(* CoDeSys 2.3 library: Flexlink V1_0.lib *)
(* Libraries: STANDARD.LIB 5.6.98 12:03:02 *)

(* Global variable list: Global_Variables *)
VAR_GLOBAL
(**************************************************************************************************************)
(* System Bit *)
(**************************************************************************************************************)

	OFF_50ms		: BOOL;
	ON_50ms		: BOOL;
	Clock50msOnPls	: BOOL;
	OFF_100ms		: BOOL;
	ON_100ms		: BOOL;
	Clock100msOnPls	: BOOL;
	OFF_500ms		: BOOL;
	ON_500ms		: BOOL;
	Clock500msOnPls	: BOOL;
	OFF_1s			: BOOL;
	ON_1s			: BOOL;
	Clock1sOnPls	: BOOL;
	Always_ON		:BOOL;
	Always_Off		:BOOL;
	Debug			:BOOL := TRUE;

(**************************************************************************************************************)
(* Machine Standard Word *)
(**************************************************************************************************************)

	ErrorDWord 			AT %MD1000:  ARRAY [0..20,1..10] OF DWORD;
	WarningDWord		AT%MD2000: ARRAY [0..20,1..10] OF DWORD;
	AutoDWord 			AT %MD3000:  ARRAY [0..20,1..10] OF DWORD;
	OriginDWord 			AT %MD4000:  ARRAY [0..20,1..10] OF DWORD;

	InputByte				AT %IB0: ARRAY [0..500] OF BYTE;
	OutputByte			AT %QB0: ARRAY [0..500] OF BYTE;

(**************************************************************************************************************)
(* Machine and Station Control *)
(**************************************************************************************************************)
	MC:Struc_Machine_Ctrl;
	SC :ARRAY[0..20] OF Struc_Station_Ctrl;

(**************************************************************************************************************)
(* Manual Control *)
(**************************************************************************************************************)
	ManualSafetyOK		:BOOL;
	M_StepFwdPls		:BOOL;
	M_StepBwdPls		:BOOL;
	M_StepRun			:BOOL;

(**************************************************************************************************************)
(* Input/Output *)
(**************************************************************************************************************)
	InputWord			AT%IB0	:ARRAY [0..100] OF BOOL;


END_VAR

(* Global variable list: Global_Variables_Error *)
VAR_GLOBAL
	E_EmgStop			: BOOL;
	E_LightCurtain		: BOOL;
	E_AirLow 			: BOOL;
	E_SafetyDoorOpen	: BOOL;
END_VAR

(* Global variable list: Global_Variables_HMI *)
VAR_GLOBAL
	T_AutoRunString:		STRING;

	T_StepRun:			BOOL;
	T_StepStop:			BOOL;
	T_StepBwd:			BOOL;
	T_StepFwd:			BOOL;
	T_StationError:		BOOL;
	T_Origin:				BOOL;
	T_OneCycleRun:		BOOL;
	T_ManualCycleTime:	TIME;
	T_Curr_Step_Station: 	UINT;
	T_EndProd:			BOOL;

	V_StepRunCurrStation:	STRING;
	V_StepRunStatus:		STRING;
	V_AutorunString:		STRING;
END_VAR

(* Global variable list: Global_Variables_Holding *)
VAR_GLOBAL RETAIN
	Password_Control: Std_Password_Ctrl;

(* Parameter Setting *)
	Number_of_Station : INT;

END_VAR

(* Data type *)
TYPE Struc_Hist_Step_Case :
STRUCT
	CurrentStepHist	: INT;
	NextStepHist		: INT;
	StepTime		: TIME;
END_STRUCT
END_TYPE

(* Data type *)
TYPE Struc_Machine_Ctrl :
STRUCT
(* Mode Bit*)
	AutoMode		:BOOL;
	ManualMode		:BOOL;

(* Status Bit*)
	DryRun			:BOOL;
	Stop			:BOOL;
	AutoRunning		:BOOL;
	StopPressed		:BOOL;


	StationStopErr 	:BOOL;
	Warning			:BOOL;
	WarningBuzzer	:BOOL;
	Trouble			:BOOL;
	ErrDetection		:BOOL;


	OriginSchRun		:BOOL;
	InxOrigin			:BOOL;
	AllOrigin			:BOOL;
	AllStationRdy		:BOOL;
	AllStationNoWP 	:BOOL;

END_STRUCT
END_TYPE

(* Data type *)
TYPE Struc_Station_Ctrl :
STRUCT

	Running			:BOOL;
	AutoRun			:BOOL;
	RunReq			:BOOL;		(*Station Start Work Request*)
	Done			:BOOL;		(*Station Work Complete*)
	RunCond		:BOOL;
	Run_NextStepPls	:BOOL;
	Run_PrevStepPls	:BOOL;
	M_Step			:BOOL;

	Origin			:BOOL;   		(* Station Already Origin *)
	Rdy				:BOOL;			(* Station Ready *)
	NoWP 			:BOOL;
	MajorFault		:BOOL;	(* Station Major Fault *)
	MinorFault		:BOOL;	(* Station Minor Fault *)
	Warning			:BOOL;		(* Station Warning *)
	Bypass			:BOOL;		(* Station Bypass *)

	Name			:STRING;
	Status			:STRING;
	CycleTime	:TIME;

END_STRUCT
END_TYPE

(* POU Password_Output, ST *)
PROGRAM Password_Output
VAR

	pls_PasswordOK: R_TRIG;
	PasswordOKPls:BOOL;
END_VAR
(**************************************************************************************************************)
(* HMI Password Control*)
(**************************************************************************************************************)

Password_Control(
	In_PasswordConfig:= '9999');

pls_PasswordOK(CLK:= Password_Control.Out_PasswordOK OR Password_Control.Out_PasswordChanged);
PasswordOKPls := pls_PasswordOK.Q;

IF PasswordOKPls THEN
	CurrentVisu := 'TP40_SETTING';
END_IF
END_PROGRAM

(* POU Std_System_Out, LD *)
PROGRAM Std_System_Out
VAR

	Clk50ms:TON;
	ClkOff50ms:TON;
	Clk100ms:TON;
	ClkOff100ms:TON;
	Clk500ms:TON;
	ClkOff500ms:TON;
	ClkOn1s:TON;
	ClkOff1s:TON;

	T50ms_RTRIG: R_TRIG;
	T100ms_RTRIG: R_TRIG;
	T500ms_RTRIG: R_TRIG;
	T1s_RTRIG: R_TRIG;

END_VAR
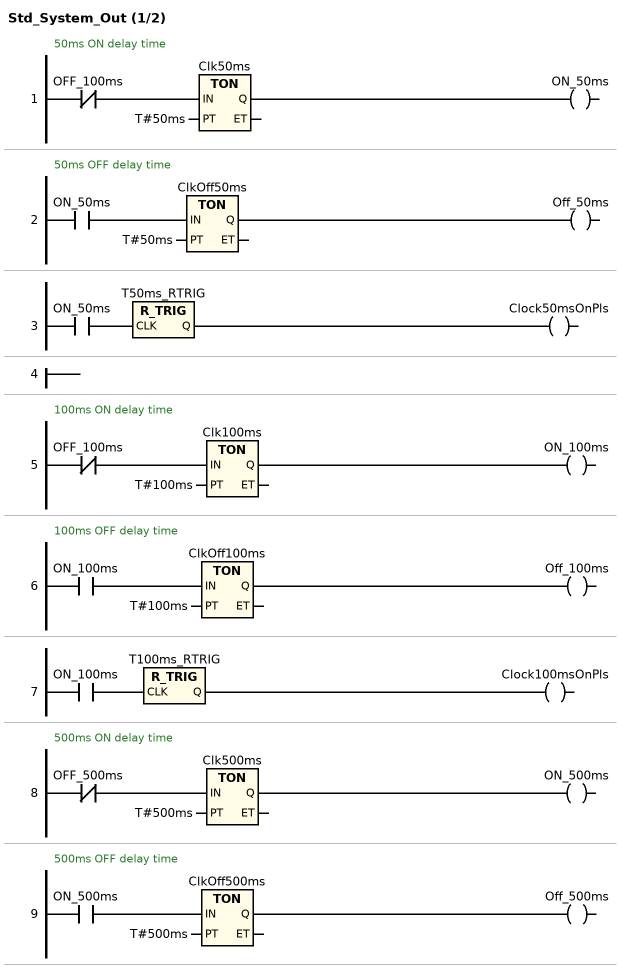
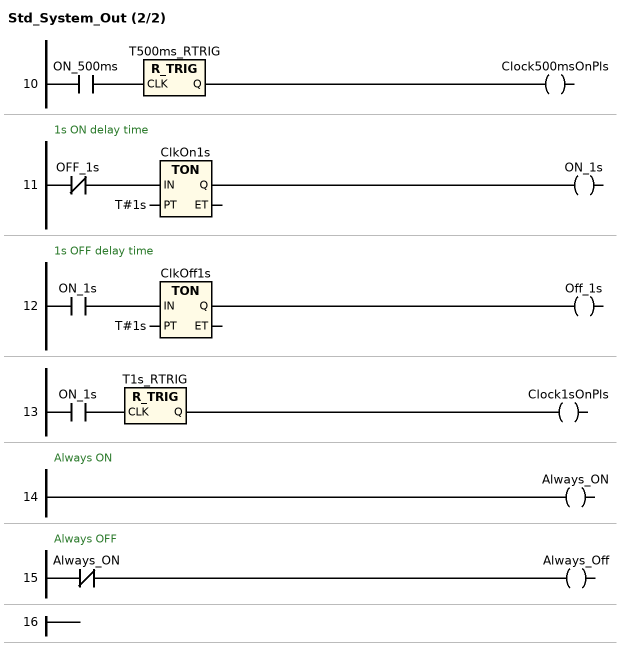
_LD_ (* Ladder Diagram *)
NETWORK 1 (* 50ms ON delay time *)
	[/OFF_100ms] - Clk50ms:TON(IN: *, PT: T#50ms) --- (ON_50ms)
NETWORK 2 (* 50ms OFF delay time *)
	[ON_50ms] - ClkOff50ms:TON(IN: *, PT: T#50ms) --- (Off_50ms)
NETWORK 3
	[ON_50ms] - T50ms_RTRIG:R_TRIG(CLK: *) --- (Clock50msOnPls)
NETWORK 4
	*
NETWORK 5 (* 100ms ON delay time *)
	[/OFF_100ms] - Clk100ms:TON(IN: *, PT: T#100ms) --- (ON_100ms)
NETWORK 6 (* 100ms OFF delay time *)
	[ON_100ms] - ClkOff100ms:TON(IN: *, PT: T#100ms) --- (Off_100ms)
NETWORK 7
	[ON_100ms] - T100ms_RTRIG:R_TRIG(CLK: *) --- (Clock100msOnPls)
NETWORK 8 (* 500ms ON delay time *)
	[/OFF_500ms] - Clk500ms:TON(IN: *, PT: T#500ms) --- (ON_500ms)
NETWORK 9 (* 500ms OFF delay time *)
	[ON_500ms] - ClkOff500ms:TON(IN: *, PT: T#500ms) --- (Off_500ms)
NETWORK 10
	[ON_500ms] - T500ms_RTRIG:R_TRIG(CLK: *) --- (Clock500msOnPls)
NETWORK 11 (* 1s ON delay time *)
	[/OFF_1s] - ClkOn1s:TON(IN: *, PT: T#1s) --- (ON_1s)
NETWORK 12 (* 1s OFF delay time *)
	[ON_1s] - ClkOff1s:TON(IN: *, PT: T#1s) --- (Off_1s)
NETWORK 13
	[ON_1s] - T1s_RTRIG:R_TRIG(CLK: *) --- (Clock1sOnPls)
NETWORK 14 (* Always ON *)
	* --- (Always_ON)
NETWORK 15 (* Always OFF *)
	[/Always_ON] --- (Always_Off)
NETWORK 16
	*
_END_LD_
(* the same logic as Structured Text *)
(* Network 1: 50ms ON delay time *)
Clk50ms(IN := NOT OFF_100ms, PT := T#50ms);
ON_50ms := Clk50ms.Q;
(* Network 2: 50ms OFF delay time *)
ClkOff50ms(IN := ON_50ms, PT := T#50ms);
Off_50ms := ClkOff50ms.Q;
(* Network 3 *)
T50ms_RTRIG(CLK := ON_50ms);
Clock50msOnPls := T50ms_RTRIG.Q;
(* Network 4 *)
(* Network 5: 100ms ON delay time *)
Clk100ms(IN := NOT OFF_100ms, PT := T#100ms);
ON_100ms := Clk100ms.Q;
(* Network 6: 100ms OFF delay time *)
ClkOff100ms(IN := ON_100ms, PT := T#100ms);
Off_100ms := ClkOff100ms.Q;
(* Network 7 *)
T100ms_RTRIG(CLK := ON_100ms);
Clock100msOnPls := T100ms_RTRIG.Q;
(* Network 8: 500ms ON delay time *)
Clk500ms(IN := NOT OFF_500ms, PT := T#500ms);
ON_500ms := Clk500ms.Q;
(* Network 9: 500ms OFF delay time *)
ClkOff500ms(IN := ON_500ms, PT := T#500ms);
Off_500ms := ClkOff500ms.Q;
(* Network 10 *)
T500ms_RTRIG(CLK := ON_500ms);
Clock500msOnPls := T500ms_RTRIG.Q;
(* Network 11: 1s ON delay time *)
ClkOn1s(IN := NOT OFF_1s, PT := T#1s);
ON_1s := ClkOn1s.Q;
(* Network 12: 1s OFF delay time *)
ClkOff1s(IN := ON_1s, PT := T#1s);
Off_1s := ClkOff1s.Q;
(* Network 13 *)
T1s_RTRIG(CLK := ON_1s);
Clock1sOnPls := T1s_RTRIG.Q;
(* Network 14: Always ON *)
Always_ON := TRUE;
(* Network 15: Always OFF *)
Always_Off := NOT Always_ON;
(* Network 16 *)
END_PROGRAM

(* POU Std_Cylinder_Ctrl, LD *)
FUNCTION_BLOCK Std_Cylinder_Ctrl

VAR_INPUT
	IN:BOOL;
	IN_CylName:STRING;
	In_Enable:BOOL;
	In_Reset:BOOL;


	(*Trigger*)
	In_AutoWork:BOOL;
	In_AutoHome:BOOL;
	In_OrgWork:BOOL;
	In_OrgHome:BOOL;
	(*Mechanical Interlock*)
	In_WorkXLock:BOOL;
	In_HomeXLock:BOOL;
	(*Sensors*)
	In_WorkRS:BOOL;
	In_HomeRS:BOOL;

	(*Timer*)
	In_WorkTON:TIME;
	In_HomeTON:TIME;
	in_Timeout:TIME;
END_VAR

VAR_OUTPUT
	Q:BOOL;
	Out_WorkSV:BOOL;
	Out_HomeSV:BOOL;
	E_WorkErr:BOOL;
	E_HomeErr:BOOL;
	S_WorkPos:BOOL;
	S_HomePos:BOOL;
END_VAR

VAR
	(* Trigger*)
	T_ManWork:BOOL;
	T_ManHome:BOOL;

	Loc_Work:BOOL;
	Loc_Home:BOOL;
	Err_Cyl:BOOL;
	Fwd_TOut: TON;
	Bwd_TOut: TON;
	Fwd_TON: TON;
	Bwd_TON: TON;
	Loc_WorkPls: BOOL;
	FwdPls: R_TRIG;
	BwdPls: R_TRIG;
	Loc_HomePls: BOOL;
	Out_RSErr:BOOL;
	FwdPosPls: F_TRIG;
	BwdPosPls: F_TRIG;
END_VAR
VAR_IN_OUT

END_VAR
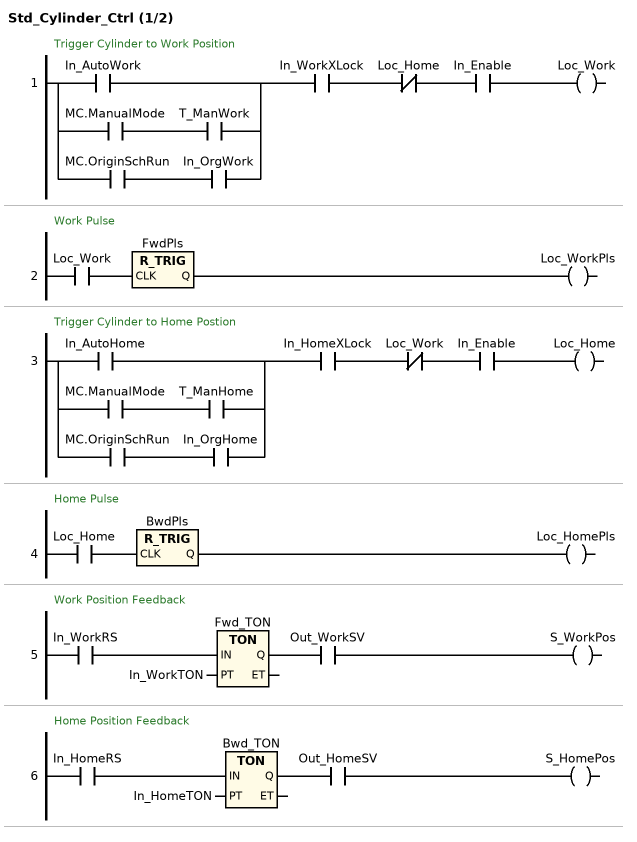
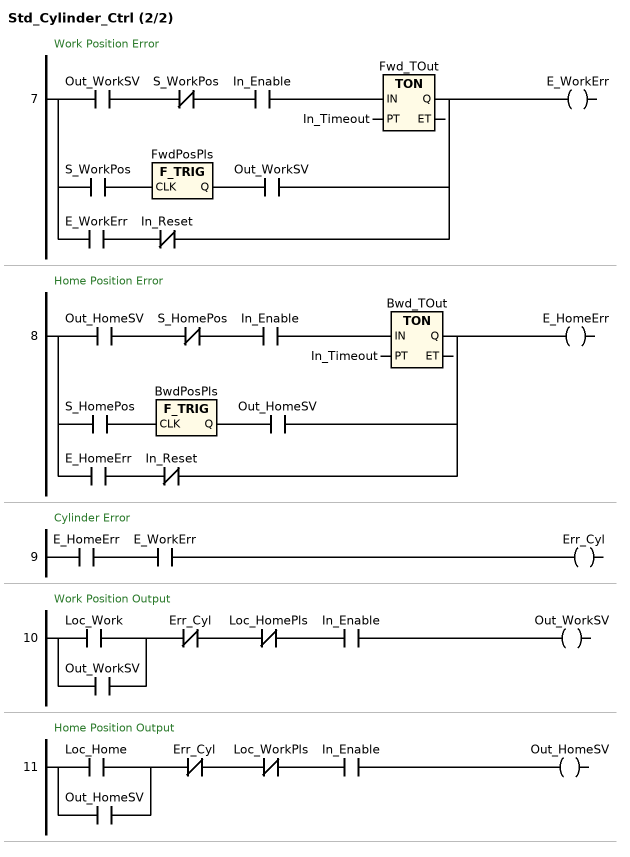
_LD_ (* Ladder Diagram *)
NETWORK 1 (* Trigger Cylinder to Work Position *)
	{ [In_AutoWork] | [MC.ManualMode] - [T_ManWork] | [MC.OriginSchRun] - [In_OrgWork] } - [In_WorkXLock] - [/Loc_Home] - [In_Enable] --- (Loc_Work)
NETWORK 2 (* Work Pulse *)
	[Loc_Work] - FwdPls:R_TRIG(CLK: *) --- (Loc_WorkPls)
NETWORK 3 (* Trigger Cylinder to Home Postion *)
	{ [In_AutoHome] | [MC.ManualMode] - [T_ManHome] | [MC.OriginSchRun] - [In_OrgHome] } - [In_HomeXLock] - [/Loc_Work] - [In_Enable] --- (Loc_Home)
NETWORK 4 (* Home Pulse *)
	[Loc_Home] - BwdPls:R_TRIG(CLK: *) --- (Loc_HomePls)
NETWORK 5 (* Work Position Feedback *)
	[In_WorkRS] - Fwd_TON:TON(IN: *, PT: In_WorkTON) - [Out_WorkSV] --- (S_WorkPos)
NETWORK 6 (* Home Position Feedback *)
	[In_HomeRS] - Bwd_TON:TON(IN: *, PT: In_HomeTON) - [Out_HomeSV] --- (S_HomePos)
NETWORK 7 (* Work Position Error *)
	{ [Out_WorkSV] - [/S_WorkPos] - [In_Enable] - Fwd_TOut:TON(IN: *, PT: In_Timeout) | [S_WorkPos] - FwdPosPls:F_TRIG(CLK: *) - [Out_WorkSV] | [E_WorkErr] - [/In_Reset] } --- (E_WorkErr)
NETWORK 8 (* Home Position Error *)
	{ [Out_HomeSV] - [/S_HomePos] - [In_Enable] - Bwd_TOut:TON(IN: *, PT: In_Timeout) | [S_HomePos] - BwdPosPls:F_TRIG(CLK: *) - [Out_HomeSV] | [E_HomeErr] - [/In_Reset] } --- (E_HomeErr)
NETWORK 9 (* Cylinder Error *)
	[E_HomeErr] - [E_WorkErr] --- (Err_Cyl)
NETWORK 10 (* Work Position Output *)
	{ [Loc_Work] | [Out_WorkSV] } - [/Err_Cyl] - [/Loc_HomePls] - [In_Enable] --- (Out_WorkSV)
NETWORK 11 (* Home Position Output *)
	{ [Loc_Home] | [Out_HomeSV] } - [/Err_Cyl] - [/Loc_WorkPls] - [In_Enable] --- (Out_HomeSV)
_END_LD_
(* the same logic as Structured Text *)
(* Network 1: Trigger Cylinder to Work Position *)
Loc_Work := (In_AutoWork OR MC.ManualMode AND T_ManWork OR MC.OriginSchRun AND In_OrgWork) AND In_WorkXLock AND NOT Loc_Home AND In_Enable;
(* Network 2: Work Pulse *)
FwdPls(CLK := Loc_Work);
Loc_WorkPls := FwdPls.Q;
(* Network 3: Trigger Cylinder to Home Postion *)
Loc_Home := (In_AutoHome OR MC.ManualMode AND T_ManHome OR MC.OriginSchRun AND In_OrgHome) AND In_HomeXLock AND NOT Loc_Work AND In_Enable;
(* Network 4: Home Pulse *)
BwdPls(CLK := Loc_Home);
Loc_HomePls := BwdPls.Q;
(* Network 5: Work Position Feedback *)
Fwd_TON(IN := In_WorkRS, PT := In_WorkTON);
S_WorkPos := Fwd_TON.Q AND Out_WorkSV;
(* Network 6: Home Position Feedback *)
Bwd_TON(IN := In_HomeRS, PT := In_HomeTON);
S_HomePos := Bwd_TON.Q AND Out_HomeSV;
(* Network 7: Work Position Error *)
Fwd_TOut(IN := Out_WorkSV AND NOT S_WorkPos AND In_Enable, PT := In_Timeout);
FwdPosPls(CLK := S_WorkPos);
E_WorkErr := Fwd_TOut.Q OR FwdPosPls.Q AND Out_WorkSV OR E_WorkErr AND NOT In_Reset;
(* Network 8: Home Position Error *)
Bwd_TOut(IN := Out_HomeSV AND NOT S_HomePos AND In_Enable, PT := In_Timeout);
BwdPosPls(CLK := S_HomePos);
E_HomeErr := Bwd_TOut.Q OR BwdPosPls.Q AND Out_HomeSV OR E_HomeErr AND NOT In_Reset;
(* Network 9: Cylinder Error *)
Err_Cyl := E_HomeErr AND E_WorkErr;
(* Network 10: Work Position Output *)
Out_WorkSV := (Loc_Work OR Out_WorkSV) AND NOT Err_Cyl AND NOT Loc_HomePls AND In_Enable;
(* Network 11: Home Position Output *)
Out_HomeSV := (Loc_Home OR Out_HomeSV) AND NOT Err_Cyl AND NOT Loc_WorkPls AND In_Enable;
END_FUNCTION_BLOCK

(* POU Std_Hist_StepCase, ST *)
FUNCTION_BLOCK Std_Hist_StepCase

VAR_INPUT
	IN:BOOL;
	CurrentStep:INT;
	NextStep:INT;
END_VAR

VAR_OUTPUT
	Q:BOOL;
	NewStep:INT;
END_VAR

VAR
	StepData:ARRAY[0..100] OF Struc_Hist_Step_Case ;

	StepTimer: TON;
	Loop: INT;
END_VAR
IF CurrentStep = NextStep THEN
StepTimer(IN:=TRUE , PT:=t#1100h , Q=> , ET=> );

StepData[0].CurrentStepHist :=CurrentStep;

ELSE
(* Copy HIstory File *)
FOR Loop := 0 TO 99 DO
StepData[100-Loop].CurrentStepHist   := StepData[99-Loop].CurrentStepHist ;
StepData[100-Loop].NextStepHist := StepData[99-Loop].NextStepHist ;
StepData[100-Loop].StepTime := StepData[99-Loop].StepTime;
END_FOR

(* Update New Data*)
StepData[1].NextStepHist:=NextStep;
StepData[1].StepTime :=StepTimer.ET;

StepTimer(IN:=FALSE , PT:=T#1100h , Q=> , ET=> );
NewStep:=NextStep;
END_IF
END_FUNCTION_BLOCK

(* POU Std_IAI_16Point, ST *)
(* @OBJECTFLAGS := '0, 8' *)
FUNCTION_BLOCK Std_IAI_16Point
VAR_INPUT
	In_Enable:BOOL;
	In_Name:STRING;
	In_AutoMode:BOOL;

	(*Trigger*)
	In_AutoStart:BOOL;
	In_OrgHome:BOOL;

	In_Pos_Num:WORD;
	In_ALM:BOOL;
	In_Reset:BOOL;
	In_PEND:BOOL;
	In_HEND:BOOL;
	In_Mec_Interlock:BOOL;
	In_PosTON:TIME;
	In_Timeout:TIME;
END_VAR

VAR_OUTPUT
	S_InPos:BOOL;  (*Current Pos*)
	S_Pos_Num : INT;
	S_InHome:BOOL;
	Out_CSTR:BOOL;
	Out_PC1:BOOL;
	Out_PC2:BOOL;
	Out_PC4:BOOL;
	Out_PC8:BOOL;
	E_Alm:BOOL;
	E_AlmPos:BOOL;
END_VAR

VAR
	(* Trigger*)
	T_ManStart:BOOL;
	T_ManHome:BOOL;
	T_ManPos_Num:INT;

	CSTR:BOOL; (*Common Start Bit*)
	Home : BOOL;
	Pos_Num:INT;

	TimePos: TON;
	BitPos1: BOOL;
	BitPos2: BOOL;
	BitPos3: BOOL;
	BitPos4: BOOL;
	TimeOut: TON;
	TempBit1: BYTE;
	TempBit2: BYTE;
	TempBit3: BYTE;
	TempBit4: BYTE;
	BytePos: BYTE;
	IAI_TimeOut: BOOL;
	Error_Alm: BOOL;
	DoneTon: BOOL;
	tmrStartDelay: TON;
	StartDelayTon: BOOL;
	plsStart: R_TRIG;
	StartDelayPls: BOOL;
	plsIAIDone: R_TRIG;
	DonePls: BOOL;
	plsHome: R_TRIG;
	HomePls: BOOL;
	HomeSearch: BOOL;
	test: BOOL;
	test1: BOOL;
	tmrStartDelay_1: TON;
	StartDelayTon_1: BOOL;
	IAI_Busy: BOOL;
	test_1: BOOL;
	tmrStartDelay_Home: TON;
	StartDelayTon_Home: BOOL;
	tmrStartDelay_Home_1: TON;
	StartDelayTon_Home_1: BOOL;
END_VAR
(**************************************************************************************************************)
(*Trigger*)
(**************************************************************************************************************)
IF  In_AutoStart OR (MC.ManualMode AND T_ManStart) THEN
CSTR := TRUE;
ELSE
CSTR := FALSE;
END_IF;

IF In_AutoMode THEN
Pos_Num := In_Pos_Num;
ELSE
Pos_Num:=T_ManPos_Num;
END_IF


IF (MC.OriginSchRun AND In_OrgHome) OR (MC.ManualMode AND T_ManHome) THEN
Home := TRUE;
Pos_Num:=0;
ELSE
Home := FALSE;
END_IF;
(**************************************************************************************************************)
(*Reset Error/Warning*)
(**************************************************************************************************************)
IF In_reset AND ( E_AlmPos OR E_Alm OR Error_Alm) THEN
	E_AlmPos :=FALSE;
	E_Alm:= FALSE;
	Error_Alm := FALSE;
END_IF;

(**************************************************************************************************************)
(*System Error*)
(**************************************************************************************************************)
(* Time Out*)
TimeOut (IN := Out_CSTR AND NOT S_InPos AND  In_Mec_Interlock, PT:=In_Timeout);
IAI_TimeOut := TimeOut.Q;

IF IAI_TimeOut AND In_Enable THEN
	E_AlmPos := TRUE;
END_IF;

(* IAI Controller Error*)
IF In_Enable AND In_ALM THEN
	E_Alm := TRUE;
END_IF;

(* IAI System In Error Condition*)
Error_Alm := E_AlmPos OR E_Alm;

IF Error_Alm THEN
	Out_CSTR := FALSE;
	S_InPos := FALSE;
	HomeSearch := FALSE;
	IAI_Busy:= FALSE;
END_IF;

(**************************************************************************************************************)
(*Moving To Target Position*)
(**************************************************************************************************************)

Out_PC1 := FALSE;
Out_PC2 := FALSE;
Out_PC4 := FALSE;
Out_PC8 := FALSE;

IF In_Enable AND NOT Error_Alm THEN
	BytePos := INT_TO_BYTE (Pos_Num);
	TempBit1 := BytePos AND 2#1;
	TempBit2 := BytePos AND 2#10;
	TempBit3 := BytePos AND 2#100;
	TempBit4 := BytePos AND 2#1000;

	BitPos1 := INT_TO_BOOL (TempBit1);
	BitPos2 := INT_TO_BOOL (TempBit2);
	BitPos3 := INT_TO_BOOL (TempBit3);
	BitPos4 := INT_TO_BOOL (TempBit4);

		IF BitPos1 THEN
			Out_PC1 := TRUE;
		END_IF;

		IF BitPos2 THEN
			Out_PC2 := TRUE;
		END_IF;

		IF BitPos3 THEN
			Out_PC4 := TRUE;
		END_IF;

		IF BitPos4 THEN
			Out_PC8 := TRUE;
		END_IF;
END_IF;

(**************************************************************************************************************)
(*Moving To Target Position Common*)
(**************************************************************************************************************)
tmrStartDelay(IN := CSTR , PT:= T#0.1s);
StartDelayTon := tmrStartDelay.Q;

plsStart(CLK := StartDelayTon);
StartDelayPls := plsStart.Q;

tmrStartDelay_1(IN := Out_CSTR , PT:= T#0.5s);
StartDelayTon_1 := tmrStartDelay_1.Q;

IF In_Enable AND NOT HomeSearch AND In_Mec_Interlock AND NOT Error_Alm THEN
	IF  StartDelayPls AND In_PEND THEN
		Out_CSTR := TRUE;
		S_InPos := FALSE;
		IAI_Busy := TRUE;
	END_IF;

	IF (StartDelayTon_1 AND Out_CSTR) OR NOT In_PEND  THEN
		Out_CSTR := FALSE;
	END_IF;
END_IF;

(**************************************************************************************************************)
(*Moving Done Complete Status*)
(**************************************************************************************************************)

TimePos (IN :=  In_PEND  AND (IAI_Busy OR HomeSearch) , PT:= In_PosTON);
DoneTon := TimePos.Q;

plsIAIDone(CLK := DoneTon);
DonePls := plsIAIDone.Q;

IF DoneTon AND In_Enable THEN
	IF HomeSearch THEN
		S_Pos_Num := 0;
	ELSE
		S_Pos_Num := Pos_Num;
	END_IF
	S_InPos := TRUE;
	HomeSearch := FALSE;
	IAI_Busy:= FALSE;
END_IF;

(**************************************************************************************************************)
(*Moving Target To Home = Pos 0*)
(**************************************************************************************************************)
S_InHome := S_Pos_Num = 0 AND S_InPos AND In_HEND;

tmrStartDelay_Home(IN := Home   , PT:= T#0.1s);
StartDelayTon_Home := tmrStartDelay_Home.Q;

plsHome (CLK:= StartDelayTon_Home AND NOT IAI_Busy );
HomePls:= plsHome.Q;

tmrStartDelay_Home_1(IN := HomeSearch AND Out_CSTR , PT:= T#0.5s);
StartDelayTon_Home_1 := tmrStartDelay_Home_1.Q;

IF In_Enable AND NOT Error_Alm AND In_Mec_Interlock AND  NOT Out_CSTR  THEN
	IF HomePls THEN
		HomeSearch := TRUE;
		Out_CSTR :=TRUE;
	END_IF;
END_IF;

IF HomeSearch AND StartDelayTon_Home_1 THEN
	Out_CSTR := FALSE;
END_IF;
END_FUNCTION_BLOCK

(* POU Std_IV_Vision_Ctrl, LD *)
FUNCTION_BLOCK Std_IV_Vision_Ctrl
VAR_INPUT
	IN: BOOL;
	In_Name:STRING;
	In_Enable:BOOL;
	In_Alm:BOOL;
	In_Reset:BOOL;
	In_AutoMode:BOOL;
	In_Auto_Model:INT;
	In_Busy:BOOL;
	In_AutoTrigger:BOOL;
	In_Result:BOOL;
	In_Timeout:TIME;
END_VAR

VAR_OUTPUT
	Q:BOOL;
	Out_ProgBit0:BOOL;
	Out_ProgBit1:BOOL;
	Out_ProgBit2:BOOL;
	Out_ProgBit3:BOOL;
	Out_Trigger:BOOL;
	Out_ClearErr:BOOL;
	S_Result:BOOL;
	S_Done:BOOL;
	E_Alm:BOOL;
END_VAR

VAR
	T_ManualTrigger:	BOOL;
	T_Manual_Model:	INT;
	Model:			INT;
	Start:			BOOL;

	TempModel: BYTE;
	ModelBit1: BYTE;
	ModelBit2: BYTE;
	ModelBit3: BYTE;
	ModelBit0: BYTE;
	TimeOut: TON;
	Reset_Result: BOOL;
	Vision_Trigger: R_TRIG;
	tmr_Done: TON;
	Start_Rtrig: R_TRIG;
END_VAR
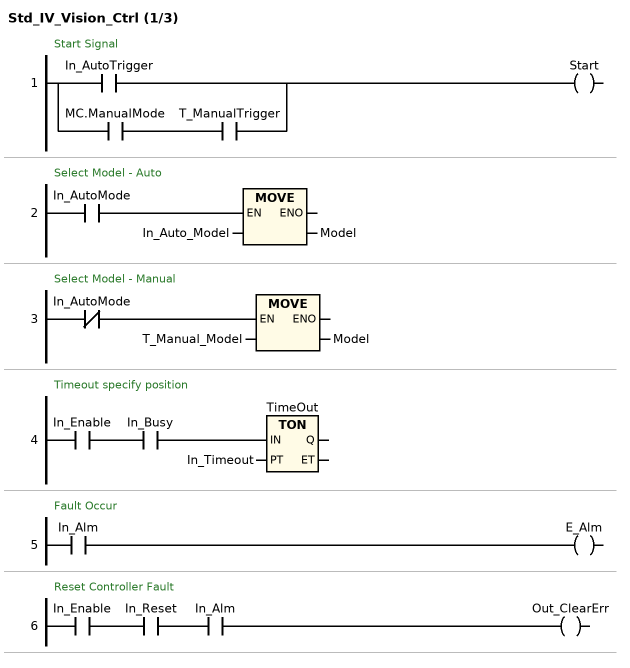
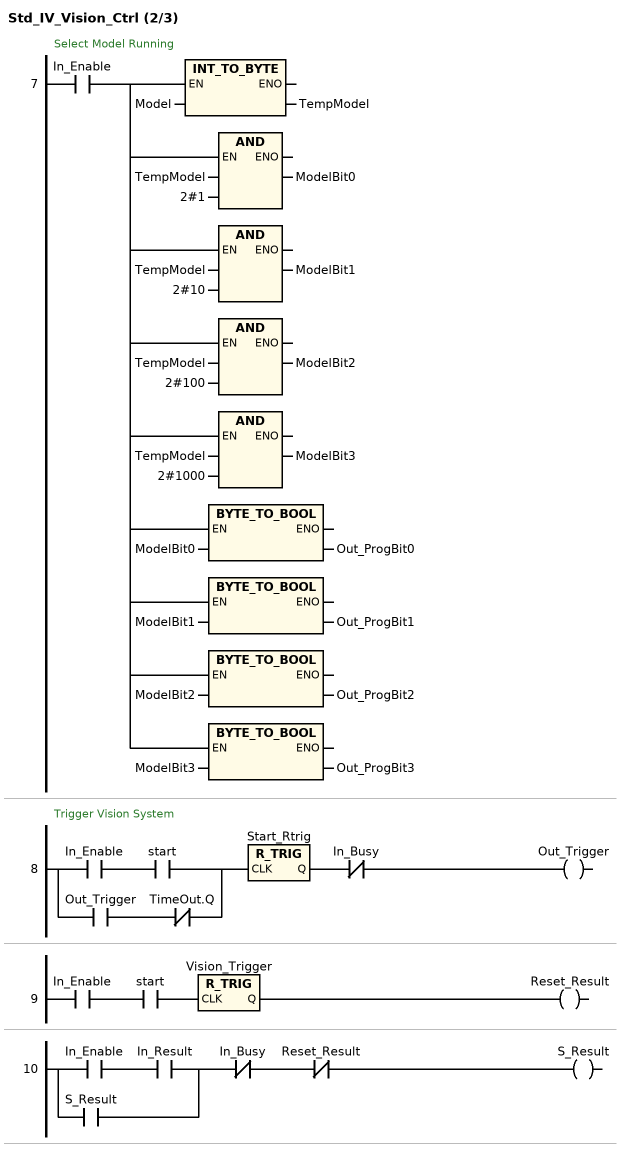
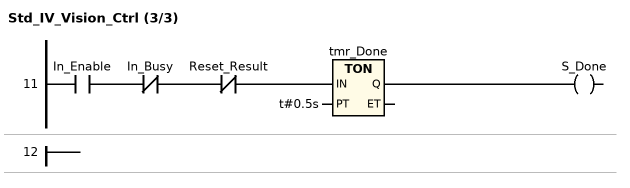
_LD_ (* Ladder Diagram *)
NETWORK 1 (* Start Signal *)
	{ [In_AutoTrigger] | [MC.ManualMode] - [T_ManualTrigger] } --- (Start)
NETWORK 2 (* Select Model - Auto *)
	[In_AutoMode]
		EN --- MOVE(In_Auto_Model) => Model
NETWORK 3 (* Select Model - Manual *)
	[/In_AutoMode]
		EN --- MOVE(T_Manual_Model) => Model
NETWORK 4 (* Timeout specify position *)
	[In_Enable] - [In_Busy] - TimeOut:TON(IN: *, PT: In_Timeout)
NETWORK 5 (* Fault Occur *)
	[In_Alm] --- (E_Alm)
NETWORK 6 (* Reset Controller Fault *)
	[In_Enable] - [In_Reset] - [In_Alm] --- (Out_ClearErr)
NETWORK 7 (* Select Model Running *)
	[In_Enable]
		EN --- INT_TO_BYTE(Model) => TempModel
		EN --- AND(TempModel, 2#1) => ModelBit0
		EN --- AND(TempModel, 2#10) => ModelBit1
		EN --- AND(TempModel, 2#100) => ModelBit2
		EN --- AND(TempModel, 2#1000) => ModelBit3
		EN --- BYTE_TO_BOOL(ModelBit0) => Out_ProgBit0
		EN --- BYTE_TO_BOOL(ModelBit1) => Out_ProgBit1
		EN --- BYTE_TO_BOOL(ModelBit2) => Out_ProgBit2
		EN --- BYTE_TO_BOOL(ModelBit3) => Out_ProgBit3
NETWORK 8 (* Trigger Vision System *)
	{ [In_Enable] - [start] | [Out_Trigger] - [/TimeOut.Q] } - Start_Rtrig:R_TRIG(CLK: *) - [/In_Busy] --- (Out_Trigger)
NETWORK 9
	[In_Enable] - [start] - Vision_Trigger:R_TRIG(CLK: *) --- (Reset_Result)
NETWORK 10
	{ [In_Enable] - [In_Result] | [S_Result] } - [/In_Busy] - [/Reset_Result] --- (S_Result)
NETWORK 11
	[In_Enable] - [/In_Busy] - [/Reset_Result] - tmr_Done:TON(IN: *, PT: t#0.5s) --- (S_Done)
NETWORK 12
	*
_END_LD_
(* the same logic as Structured Text *)
(* Network 1: Start Signal *)
Start := In_AutoTrigger OR MC.ManualMode AND T_ManualTrigger;
(* Network 2: Select Model - Auto *)
IF In_AutoMode THEN
	Model := In_Auto_Model;
END_IF;
(* Network 3: Select Model - Manual *)
IF NOT In_AutoMode THEN
	Model := T_Manual_Model;
END_IF;
(* Network 4: Timeout specify position *)
TimeOut(IN := In_Enable AND In_Busy, PT := In_Timeout);
(* Network 5: Fault Occur *)
E_Alm := In_Alm;
(* Network 6: Reset Controller Fault *)
Out_ClearErr := In_Enable AND In_Reset AND In_Alm;
(* Network 7: Select Model Running *)
IF In_Enable THEN
	TempModel := INT_TO_BYTE(Model);
	ModelBit0 := TempModel AND 2#1;
	ModelBit1 := TempModel AND 2#10;
	ModelBit2 := TempModel AND 2#100;
	ModelBit3 := TempModel AND 2#1000;
	Out_ProgBit0 := BYTE_TO_BOOL(ModelBit0);
	Out_ProgBit1 := BYTE_TO_BOOL(ModelBit1);
	Out_ProgBit2 := BYTE_TO_BOOL(ModelBit2);
	Out_ProgBit3 := BYTE_TO_BOOL(ModelBit3);
END_IF;
(* Network 8: Trigger Vision System *)
Start_Rtrig(CLK := In_Enable AND start OR Out_Trigger AND NOT TimeOut.Q);
Out_Trigger := Start_Rtrig.Q AND NOT In_Busy;
(* Network 9 *)
Vision_Trigger(CLK := In_Enable AND start);
Reset_Result := Vision_Trigger.Q;
(* Network 10 *)
S_Result := (In_Enable AND In_Result OR S_Result) AND NOT In_Busy AND NOT Reset_Result;
(* Network 11 *)
tmr_Done(IN := In_Enable AND NOT In_Busy AND NOT Reset_Result, PT := t#0.5s);
S_Done := tmr_Done.Q;
(* Network 12 *)
END_FUNCTION_BLOCK

(* POU Std_Machine_Ctrl, ST *)
FUNCTION_BLOCK Std_Machine_Ctrl

VAR_INPUT
	In_Start_PB:						BOOL;
	In_Stop_PB:						BOOL;
	In_EmgOK:						BOOL;
	In_Door_Sw: 						BOOL;
	In_Pressure_Sw: 					BOOL;
	In_LightCurtainSafeToCross:		BOOL;
	In_LightCurtainOK: 					BOOL;
	In_OtherTrouble: 					BOOL;
	In_Reset_PB:						BOOL;
	In_Start_Enable:					BOOL;
	In_EndProdWPCleared:			BOOL;
	I_StepFwdPB:					BOOL;
	I_StepBwdPB:					BOOL;

END_VAR

VAR_IN_OUT

END_VAR

VAR_OUTPUT
	Out_RedTower:BOOL;
	Out_YelTower :BOOL;
	Out_GrnTower:BOOL;
	Out_Buzzer:BOOL;

END_VAR

VAR
	Loop: INT;
	LoopStation: INT;
(*************************************************************************************************************************************)
(*Status Bit*)
(*************************************************************************************************************************************)

	AllStationStop:BOOL;

(*************************************************************************************************************************************)
(* HMI Bit*)
(*************************************************************************************************************************************)
	T_Auto: 				BOOL;
	T_Manual:			BOOL;
	T_DryRun: 			BOOL;
	T_OriginSearch:		BOOL;
	T_Start:				BOOL;
	T_Stop:				BOOL;
	T_Reset :			BOOL;
 	T_Station_BypassP: 	ARRAY [0..50] OF BOOL;
	T_BypassDoor: 		BOOL;
	T_BypassBuzzer:		BOOL;
	T_BuzzerOff :			BOOL;
	T_AutoMsgAlarm: 		BOOL;
	T_StatusString: 		STRING;
	V_AutorunString: 		STRING;
(*************************************************************************************************************************************)
(*Auto*)
(*************************************************************************************************************************************)
	AutoPBMem: BOOL;
	NotAutoRunning:BOOL;

	pls_OriginSchRun: R_TRIG;
	OriginSchRunPls: BOOL;

(*************************************************************************************************************************************)
(*Manual*)
(*************************************************************************************************************************************)
	Pls_StepFwd: 	R_TRIG;
	Pls_StepBwd: 	R_TRIG;
	CycleTimer: 		TON;
	ManualCond: 		BOOL;
(*************************************************************************************************************************************)
	(* Error Handling*)
(*************************************************************************************************************************************)

	tmrEmgOn: TON;
	EmgPBTON :BOOL;

	tmrEmgOn_Air: TON;
	EmgPBTON_Air: BOOL;

	Reset:BOOL;
	pls_Reset :R_TRIG;
	ResetPls:BOOL;

	tmrDoorSwitch: TON;
	DoorSwTOFF: BOOL;

	tmrCurtainCrossed: TON;
	CurtainCrossedTON:BOOL;


END_VAR
(**************************************************************************************************************)
(* Auto Mode Selection*)
(**************************************************************************************************************)
IF T_Auto THEN
	AutoPBMem := TRUE;
END_IF;

IF( AutoPBMem OR MC.AutoRunning) AND NOT MC.Trouble THEN
	MC.AutoMode := TRUE;
ELSE
	MC.AutoMode := FALSE;
	AutoPBMem := FALSE;
END_IF;


(**************************************************************************************************************)
(*Manual Mode Selection*)
(**************************************************************************************************************)
IF T_Manual THEN
	AutoPBMem := FALSE;
END_IF;

IF NOT (AutoPBMem OR MC.AutoRunning OR MC.Trouble) THEN
	MC.ManualMode :=TRUE;
ELSE
	MC.ManualMode :=FALSE;
END_IF;


(**************************************************************************************************************)
(* Manual Interlocking *)
(**************************************************************************************************************)

ManualSafetyOK 	:=TRUE;
ManualCond 		:= MC.ManualMode AND ManualSafetyOK AND NOT mc.OriginSchRun;

(**************************************************************************************************************)
(* Manual General*)
(**************************************************************************************************************)

Pls_StepFwd(CLK:= I_StepFwdPB OR T_StepFwd);
M_StepFwdPls := Pls_StepFwd.Q;

Pls_StepBwd(CLK:= I_StepBwdPB OR T_StepBwd);
M_StepBwdPls := Pls_StepBwd.Q;


(**************************************************************************************************************)
(* Manual Stepping Mode*)
(**************************************************************************************************************)
IF (NOT T_StepStop) AND ManualCond THEN
	IF T_StepRun THEN
		M_StepRun := TRUE;
	END_IF;
ELSE
		M_StepRun := FALSE;
END_IF;


(* Display Status on Visio*)
T_StationError 		:= sc[T_Curr_Step_Station].MajorFault OR sc[T_Curr_Step_Station].MinorFault;
T_Origin 				:=sc[T_Curr_Step_Station].Origin;
V_StepRunCurrStation 	:= sc[T_Curr_Step_Station].Name;
V_StepRunStatus 		:= sc[T_Curr_Step_Station].Status;


FOR Loop := 1 TO Number_of_Station BY 1 DO
SC[Loop].M_Step		:= FALSE;
END_FOR

IF M_StepRun THEN
SC[T_Curr_Step_Station].M_Step	:= TRUE;
END_IF;


(* CycleTime Calculation*)
CycleTimer(IN:=M_StepRun , PT:=t#1100h , Q=> , ET=> );

IF M_StepRun THEN
T_ManualCycleTime :=CycleTimer.ET;
END_IF


(**************************************************************************************************************)
(*Reset Auto and Origin Bit*)
(**************************************************************************************************************)
	FOR LoopStation := 0 TO 20 BY 1 DO
		IF NOT (SC[LoopStation].AutoRun OR SC[LoopStation].M_Step OR MC.AutoMode)  THEN
			FOR Loop := 1 TO 10 BY 1 DO
				AutoDWord[LoopStation,Loop] :=0;
			END_FOR
		END_IF
	END_FOR

	FOR LoopStation := 0 TO 20 BY 1 DO
		IF NOT MC.OriginSchRun THEN
			FOR Loop := 1 TO 10 BY 1 DO
				OriginDWord[LoopStation,Loop] :=0;
			END_FOR
		END_IF
	END_FOR

(**************************************************************************************************************)
(*Origin Search Run*)
(**************************************************************************************************************)
IF MC.ManualMode AND NOT MC.AllOrigin AND NOT (MC.StationStopErr OR MC.Trouble OR MC.StopPressed )  THEN
	IF T_OriginSearch THEN
		MC.OriginSchRun  := TRUE;
	END_IF;
ELSE
	MC.OriginSchRun := FALSE;
END_IF;

pls_OriginSchRun(CLK:= MC.OriginSchRun);
OriginSchRunPls := pls_OriginSchRun.Q;


(**************************************************************************************************************)
(*Dry Run Mode Selection*)
(**************************************************************************************************************)
IF NOT MC.AutoRunning AND T_DryRun THEN
	MC.DryRun := TRUE;
END_IF;

IF NOT MC.AutoRunning AND NOT T_DryRun THEN
	MC.DryRun := FALSE;
	T_EndProd := FALSE;
END_IF;


(**************************************************************************************************************)
(* Machine Start *)
(**************************************************************************************************************)
IF MC.AutoMode AND NOT MC.Stop THEN
	IF (In_Start_PB OR T_Start) AND
		NOT MC.StationStopErr AND In_Start_Enable THEN
		MC.AutoRunning := TRUE;
	END_IF;
ELSE
	MC.AutoRunning := FALSE;
END_IF;

NotAutoRunning := NOT MC.AutoRunning;

IF MC.AutoRunning THEN
	V_AutorunString := 'Running';
ELSE
	V_AutorunString := 'Auto Mode';
END_IF


(**************************************************************************************************************)
(* Machine Stop *)
(**************************************************************************************************************)
IF MC.AutoRunning THEN
	IF NOT In_Stop_PB OR T_Stop OR In_EndProdWPCleared OR MC.StationStopErr THEN
		MC.StopPressed := TRUE;
	END_IF;
ELSE
	MC.StopPressed := FALSE;
END_IF;

IF MC.StopPressed AND AllStationStop THEN
	MC.Stop:=TRUE;
ELSE
	MC.Stop :=FALSE;
END_IF;


(**************************************************************************************************************)
(* Machine Status *)
(*From Station Status*)
(**************************************************************************************************************)

FOR Loop := 0 TO Number_of_Station BY 1  DO
IF NOT SC[Loop].Running THEN
AllStationStop := TRUE;
ELSE
AllStationStop := FALSE;
EXIT;
END_IF
END_FOR

FOR Loop := 0 TO Number_of_Station BY 1  DO
IF SC[Loop].Rdy THEN
MC.AllStationRdy := TRUE;
ELSE
MC.AllStationRdy := FALSE;
EXIT;
END_IF
END_FOR


FOR Loop := 0 TO Number_of_Station BY 1  DO
IF SC[Loop].NoWP THEN
MC.AllStationNoWP := TRUE;
ELSE
MC.AllStationNoWP := FALSE;
EXIT;
END_IF
END_FOR


FOR Loop := 0 TO Number_of_Station BY 1  DO
IF SC[Loop].Origin THEN
MC.AllOrigin:= TRUE;
ELSE
MC.AllOrigin := FALSE;
EXIT;
END_IF
END_FOR


(*Major Error for Immediate Stop*)
MC.Trouble:=E_EmgStop OR E_AirLow OR E_LightCurtain ;


FOR Loop := 0 TO Number_of_Station BY 1  DO
IF SC[Loop].MajorFault THEN
MC.Trouble:= TRUE;
END_IF
END_FOR

(*Minor Error for Stop after one cycle*)
MC.StationStopErr := E_SafetyDoorOpen  OR E_LightCurtain;

FOR Loop := 0 TO Number_of_Station BY 1  DO
IF SC[Loop].MinorFault THEN
MC.StationStopErr:= TRUE;
END_IF
END_FOR

(**************************************************************************************************************)
(* Auto Msg Alarm Display  *)
(**************************************************************************************************************)

IF MC.Trouble THEN
	T_StatusString := 'Machine Major Error';
ELSIF MC.StationStopErr THEN
	T_StatusString := 'Machine Station Error';
ELSIF MC.AutoMode THEN
	T_StatusString := 'Auto Mode';
ELSIF MC.ManualMode THEN
	T_StatusString := 'Manual Mode';
ELSIF MC.AutoRunning THEN
	T_StatusString := 'Auto Running';
END_IF

(**************************************************************************************************************)
(* For programmer Station Bypass - Debug Only*)
(**************************************************************************************************************)
IF NOT  MC.AutoRunning THEN

FOR Loop := 0 TO 20 DO
	IF T_Station_BypassP[Loop] THEN
            SC[Loop].Bypass := TRUE;
	ELSE
	    SC[Loop].Bypass := FALSE;
      END_IF;
END_FOR

END_IF;


(*************************************************************************************************************************************)
(* Reset Error And Warning Memory*)
(*************************************************************************************************************************************)

tmrEmgOn (IN := In_EmgOK, pt := T#1s);
EmgPBTON := tmrEmgOn.Q;

tmrEmgOn_Air (IN := In_EmgOK, pt := T#3s);
EmgPBTON_Air := tmrEmgOn_Air.Q;

Reset := T_Reset OR In_Reset_PB;

pls_Reset (CLK := Reset);
ResetPls := pls_Reset.Q;

(* Reset Error*)
	IF ResetPls AND EmgPBTON THEN
	FOR LoopStation := 0 TO 20 BY 1 DO
		FOR Loop := 1 TO 10 BY 1 DO
			ErrorDWord[LoopStation,Loop] :=0;
			WarningDWord[LoopStation,Loop] :=0;
		END_FOR
	END_FOR

			E_EmgStop:=FALSE;
			E_LightCurtain:=FALSE;
			E_AirLow :=FALSE;
			E_SafetyDoorOpen:=FALSE;

	END_IF;

(* Set Warning*)
MC.Warning := FALSE;
FOR LoopStation := 0 TO 20 BY 1 DO
	FOR Loop := 1 TO 10 DO
		IF WarningDWord[LoopStation,Loop]>0  THEN
			MC.Warning := TRUE;
		END_IF;
	END_FOR
END_FOR

T_AutoMsgAlarm := MC.Trouble OR MC.StationStopErr OR (NOT MC.AutoRunning AND NOT MC.AllOrigin) ;
(*************************************************************************************************************************************)
(*Error And Warning Summaries*)
(*************************************************************************************************************************************)
MC.ErrDetection := MC.AutoRunning OR MC.OriginSchRun;

(*************************************************************************************************************************************)
(*General Error and Trouble*)
(*************************************************************************************************************************************)

(*E-stop Error*)
IF NOT EmgPBTON THEN
	E_EmgStop := TRUE;
END_IF;

(*Safety Door Error*)
tmrDoorSwitch (in:= NOT In_Door_Sw, PT:= t#0.2S);
DoorSwTOFF := tmrDoorSwitch.Q;

IF MC.AutoMode AND DoorSwTOFF AND NOT T_BypassDoor THEN
	E_SafetyDoorOpen := TRUE;
END_IF;

(*Air Low Error*)
IF EmgPBTON_Air AND NOT In_Pressure_Sw THEN
	E_AirLow := TRUE;
END_IF;

(*Light Curtain Crossed Error*)
tmrCurtainCrossed(IN := NOT In_LightCurtainOK, PT:= t#0.1s);
CurtainCrossedTON := tmrCurtainCrossed.Q;

IF NOT In_LightCurtainSafeToCross  AND NOT In_LightCurtainOK THEN
	E_LightCurtain := TRUE;
END_IF;

(**************************************************************************************************************)
(* General Output*)
(**************************************************************************************************************)

Out_RedTower := MC.Trouble OR ( MC.StationStopErr AND ON_1s);

Out_YelTower :=  MC.ManualMode OR ( MC.Warning AND ON_1s AND NOT  MC.Trouble AND NOT  MC.StationStopErr );

Out_GrnTower := (MC.AutoRunning AND NOT MC.StopPressed) OR (MC.StopPressed AND ON_1s);

IF NOT (Out_RedTower OR MC.Warning) THEN
	T_BuzzerOff := FALSE;
END_IF

Out_Buzzer := (Out_RedTower OR (MC.Warning AND ON_1s)) AND NOT T_BuzzerOff AND NOT T_BypassBuzzer;
END_FUNCTION_BLOCK

(* POU Std_OnOffDev_Ctrl, LD *)
FUNCTION_BLOCK Std_OnOffDev_Ctrl

VAR_INPUT
	IN:BOOL;
	IN_DevName:STRING;
	In_Enable:BOOL;
	In_Reset:BOOL;


	(*Trigger*)
	In_AutoON:BOOL;
	In_OrgON:BOOL;

	(*Mechanical Interlock*)
	In_OnXLock:BOOL;

	(*Sensors*)
	In_ONSig:BOOL;

	(*Timer*)
	In_OnTON:TIME;
	in_Timeout:TIME;

END_VAR

VAR_OUTPUT
	Q:BOOL;
	Out_OnSV:BOOL;
	E_OnErr:BOOL;
	S_OnSig:BOOL;

END_VAR

VAR
	(* Trigger*)
	T_ManOn:BOOL;
	T_ManOff:BOOL;

	Loc_On:BOOL;
	On_TOut: TON;
	On_TON: TON;
	Loc_OnPls: BOOL;
	OnPls: R_TRIG;
	Out_RSErr:BOOL;
	OnPosPls: F_TRIG;

END_VAR
VAR_IN_OUT

END_VAR
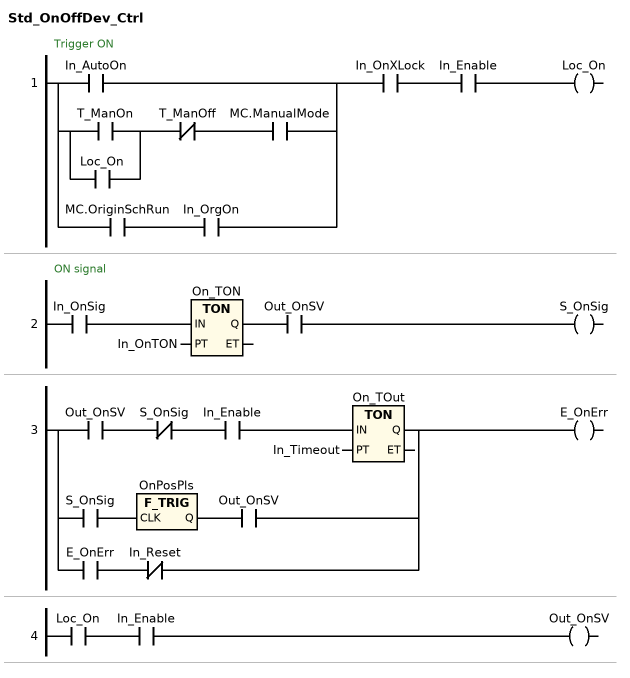
_LD_ (* Ladder Diagram *)
NETWORK 1 (* Trigger ON *)
	{ [In_AutoOn] | { [T_ManOn] | [Loc_On] } - [/T_ManOff] - [MC.ManualMode] | [MC.OriginSchRun] - [In_OrgOn] } - [In_OnXLock] - [In_Enable] --- (Loc_On)
NETWORK 2 (* ON signal *)
	[In_OnSig] - On_TON:TON(IN: *, PT: In_OnTON) - [Out_OnSV] --- (S_OnSig)
NETWORK 3
	{ [Out_OnSV] - [/S_OnSig] - [In_Enable] - On_TOut:TON(IN: *, PT: In_Timeout) | [S_OnSig] - OnPosPls:F_TRIG(CLK: *) - [Out_OnSV] | [E_OnErr] - [/In_Reset] } --- (E_OnErr)
NETWORK 4
	[Loc_On] - [In_Enable] --- (Out_OnSV)
_END_LD_
(* the same logic as Structured Text *)
(* Network 1: Trigger ON *)
Loc_On := (In_AutoOn OR (T_ManOn OR Loc_On) AND NOT T_ManOff AND MC.ManualMode OR MC.OriginSchRun AND In_OrgOn) AND In_OnXLock AND In_Enable;
(* Network 2: ON signal *)
On_TON(IN := In_OnSig, PT := In_OnTON);
S_OnSig := On_TON.Q AND Out_OnSV;
(* Network 3 *)
On_TOut(IN := Out_OnSV AND NOT S_OnSig AND In_Enable, PT := In_Timeout);
OnPosPls(CLK := S_OnSig);
E_OnErr := On_TOut.Q OR OnPosPls.Q AND Out_OnSV OR E_OnErr AND NOT In_Reset;
(* Network 4 *)
Out_OnSV := Loc_On AND In_Enable;
END_FUNCTION_BLOCK

(* POU Std_Password_Ctrl, ST *)
(* @OBJECTFLAGS := '0, 8' *)
FUNCTION_BLOCK Std_Password_Ctrl
VAR_INPUT
	In_PasswordConfig:STRING;
	In_SelectedPasswordLvl:INT; (* 0   - operator, 1 - Supervisor, 3-Maintenance *)
END_VAR
VAR_OUTPUT

END_VAR
VAR RETAIN
	In_EntryPasswordString:STRING;
	In_NewPasswordString1:STRING;
	In_NewPasswordString2:STRING;
	In_CurrPasswordStringOperator:STRING;
	In_CurrPasswordStringSupervisor:STRING;
	In_CurrPasswordStringMaintenance:STRING;
	In_EnterPassword:BOOL;
	In_ChangePassword:BOOL;

	Out_PasswordOK:BOOL;
	Out_PasswordChanged:BOOL;
	Out_CurrPasswordString:STRING;
	Out_StatusString:STRING;
	Out_PasswordConfig:BOOL;
	Out_CurrentPasswordLvl:INT; (* 0   - operator, 1 - Supervisor, 3-Maintenance *)

	PasswordOK:BOOL;
	tmrStatusChanged: TON;
	StatusChanged: BOOL;
	StatusChangedTON: BOOL;

	PaswordEnteredPls:BOOL;
	pls_PasswordEntered:R_TRIG;
	NewPaswordEnteredPls:BOOL;
	pls_NewPasswordEntered:R_TRIG;

END_VAR
tmrStatusChanged(IN := StatusChanged, PT:= t#2s);
StatusChangedTON := tmrStatusChanged.Q;

pls_PasswordEntered(CLK:= In_EnterPassword);
PaswordEnteredPls := pls_PasswordEntered.Q;

pls_NewPasswordEntered(CLK:= In_ChangePassword);
NewPaswordEnteredPls := pls_NewPasswordEntered.Q;

IF StatusChangedTON THEN
	Out_StatusString := '';
	StatusChanged := FALSE;
END_IF

(************************************************************************************************)
(* Password Entry*)
(************************************************************************************************)

IF PaswordEnteredPls THEN
	IF (In_EntryPasswordString =In_CurrPasswordStringOperator AND In_SelectedPasswordLvl =0) OR
	(In_EntryPasswordString =In_CurrPasswordStringSupervisor AND In_SelectedPasswordLvl =1) OR
	(In_EntryPasswordString =In_CurrPasswordStringMaintenance AND In_SelectedPasswordLvl =2)  THEN
		Out_PasswordOK := TRUE;
		PasswordOK := TRUE;
		Out_PasswordConfig := FALSE;
		Out_StatusString := 'Password OK!';
		Out_CurrentPasswordLvl:=In_SelectedPasswordLvl;
	ELSIF In_EntryPasswordString = In_PasswordConfig THEN
		Out_PasswordOK := TRUE;
		Out_PasswordConfig := TRUE;
		PasswordOK := TRUE;
		Out_StatusString := 'Password Config OK!';
	ELSE
		Out_PasswordConfig := FALSE;
		Out_StatusString := 'Wrong Password!';
	END_IF
	StatusChanged := TRUE;
ELSE
	Out_PasswordOK := FALSE;
END_IF



(************************************************************************************************)
(* Password Change*)
(************************************************************************************************)

IF NewPaswordEnteredPls  THEN
	IF( In_EntryPasswordString = In_CurrPasswordStringMaintenance) OR In_SelectedPasswordLvl < 2 THEN
		IF In_NewPasswordString1 <> '' AND In_NewPasswordString2 <>''  THEN
			IF In_NewPasswordString1 = In_NewPasswordString2 THEN
					CASE In_SelectedPasswordLvl OF
						0: In_CurrPasswordStringOperator :=In_NewPasswordString1;
						1: In_CurrPasswordStringSupervisor :=In_NewPasswordString1;
						2: In_CurrPasswordStringMaintenance :=In_NewPasswordString1;
					END_CASE
				Out_PasswordChanged := TRUE;
				Out_StatusString := 'Password Changed!';
			ELSE
				Out_StatusString := 'New Passwords not match!';
			END_IF
		ELSE
			Out_StatusString := 'New Password is empty!';
		END_IF
	ELSE
		Out_StatusString := 'Old Password is wrong!';
	END_IF
	StatusChanged := TRUE;
ELSE
	Out_PasswordChanged := FALSE;
END_IF

(* Reset password String *)
IF PaswordEnteredPls OR NewPaswordEnteredPls THEN
	In_EntryPasswordString :='';
	In_NewPasswordString1:='';
	In_NewPasswordString2:='';
END_IF
END_FUNCTION_BLOCK

(* POU Std_StepCase, ST *)
FUNCTION_BLOCK Std_StepCase

VAR_INPUT
	IN:BOOL;
	Step_Number: INT;
END_VAR
VAR_OUTPUT
	Q: BOOL;
	Step: ARRAY [0..9999] OF BOOL;
END_VAR

VAR
	Loop: INT;
END_VAR
FOR  Loop := 0 TO 9999 DO

IF Step_Number = Loop  THEN
Step[Loop] :=TRUE;
ELSE
Step[Loop] := FALSE;
END_IF

END_FOR
END_FUNCTION_BLOCK

(* Visualisation Blue_Ind
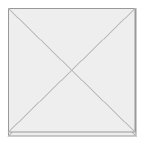
bitmap at (0,0)-(128,128): c:\flexlink\bitmap\button_blank_blue_01.bmp
bitmap at (0,0)-(127,124): c:\flexlink\bitmap\\button_blank_gray_01.bmp
*)

(* Visualisation ButtonGreenInd
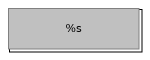
rectangle at (0,0)-(131,41): text "%s"; shows $Text$; alarm colour if $ColourTag$; taps $TapTag$; runs INTERN ASSIGN $ValueTag$:=($AssignValue$)
1 more shapes without text or variables
*)

(* Visualisation Green_Ind
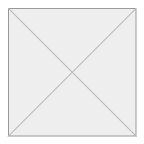
bitmap at (0,0)-(128,128): c:\flexlink\bitmap\button_blank_gray_01.bmp
bitmap at (0,0)-(128,128): c:\flexlink\bitmap\button_blank_green_01.bmp
*)

(* Visualisation IO_Monitor
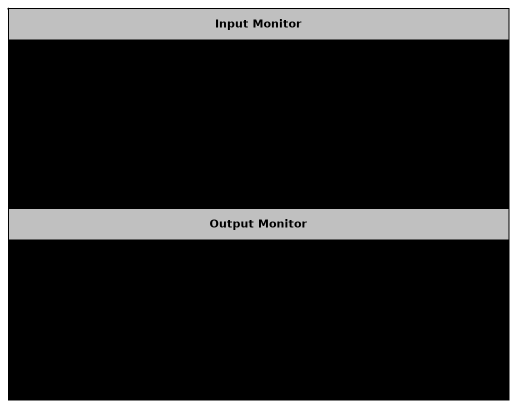
rectangle at (0,0)-(0,0): alarm colour if InputByte[INDEX].7
rectangle at (0,0)-(0,0): alarm colour if InputByte[INDEX].6
rectangle at (0,0)-(0,0): alarm colour if InputByte[INDEX].5
rectangle at (0,0)-(0,0): alarm colour if InputByte[INDEX].4
rectangle at (0,0)-(0,0): alarm colour if InputByte[INDEX].3
rectangle at (0,0)-(0,0): alarm colour if InputByte[INDEX].2
rectangle at (0,0)-(0,0): alarm colour if InputByte[INDEX].1
rectangle at (0,0)-(0,0): alarm colour if InputByte[INDEX].0
rectangle at (0,0)-(501,32): text "Input Monitor"
rectangle at (0,0)-(0,0): alarm colour if OutputByte[INDEX].7
rectangle at (0,0)-(0,0): alarm colour if OutputByte[INDEX].6
rectangle at (0,0)-(0,0): alarm colour if OutputByte[INDEX].5
rectangle at (0,0)-(0,0): alarm colour if OutputByte[INDEX].4
rectangle at (0,0)-(0,0): alarm colour if OutputByte[INDEX].3
rectangle at (0,0)-(0,0): alarm colour if OutputByte[INDEX].2
rectangle at (0,0)-(0,0): alarm colour if OutputByte[INDEX].1
rectangle at (0,0)-(0,0): alarm colour if OutputByte[INDEX].0
rectangle at (0,200)-(501,232): text "Output Monitor"
1 more shapes without text or variables
*)

(* Visualisation MANUAL_STEP
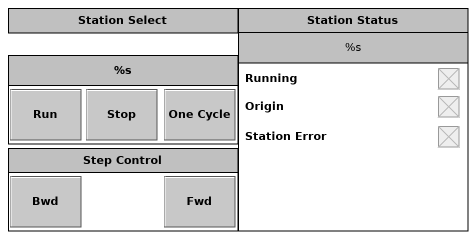
rectangle at (0,47)-(230,78): text "%s"; shows .V_StepRunCurrStation
rounded rectangle at (20,-3)-(209,28): text "Station Select"
button at (2,81)-(73,132): text "Run"; taps .T_StepRun
button at (78,81)-(149,132): text "Stop"; taps .T_StepStop
button at (156,81)-(227,132): text "One Cycle"; toggles .T_OneCycleRun
rounded rectangle at (20,137)-(209,168): text "Step Control"
button at (2,168)-(73,219): text "Bwd"; taps .T_StepBwd
button at (156,168)-(227,219): text "Fwd"; taps .T_StepFwd
rounded rectangle at (250,-3)-(439,28): text "Station Status"
rounded rectangle at (235,55)-(331,86): text "Running"
rounded rectangle at (235,83)-(331,114): text "Origin"
rounded rectangle at (235,113)-(331,144): text "Station Error"
rectangle at (230,24)-(460,55): text "%s"; shows V_StepRunStatus
embedded screen at (430,118)-(451,139): Red_Ind
embedded screen at (430,88)-(451,109): Green_Ind
embedded screen at (430,60)-(451,81): Green_Ind
6 more shapes without text or variables
1 elements of other kinds (tables, trends, ...) not read
*)

(* Visualisation Red_Ind
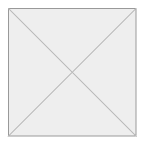
bitmap at (0,0)-(128,128): c:\flexlink\bitmap\button_blank_gray_01.bmp
bitmap at (0,0)-(128,128): c:\flexlink\bitmap\button_blank_red_01.bmp
*)

(* Visualisation Std_Alm_Ctrl_Button
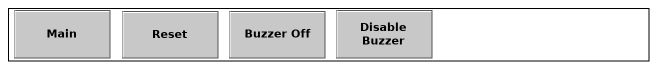
button at (6,1)-(102,49): text "Main"; opens TP00_MAIN
button at (114,2)-(210,49): text "Reset"; taps $Inst$.T_Reset
rectangle at (229,2)-(310,48): text "Buzzer Off"; alarm colour if .T_BuzzerOff; toggles $Inst$.T_BuzzerOff
rectangle at (330,4)-(421,46): text "Disable / Buzzer"; alarm colour if .T_BypassBuzzer; toggles $Inst$.T_BypassBuzzer
3 more shapes without text or variables
*)

(* Visualisation Std_Cylinder_Ctrl
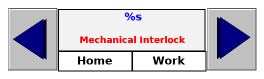
rounded rectangle at (48,0)-(195,42): text "%s"; shows $Inst$.IN_CylName
rounded rectangle at (48,42)-(122,62): text "Home"; invisible if $Inst$.E_HomeErr; alarm colour if $Inst$.S_HomePos
rounded rectangle at (122,42)-(196,62): text "Work"; invisible if $Inst$.E_WorkErr; alarm colour if $Inst$.S_WorkPos
group at (-2,-1)-(47,61)
  button at (0,0)-(49,62): taps $Inst$.In_ManHome
group at (197,-1)-(246,61)
  button at (0,0)-(49,61): taps $Inst$.In_ManWork
rounded rectangle at (49,21)-(196,41): text "Mechanical Interlock"; invisible if NOT (NOT $Inst$.In_WorkXLock AND $Inst$.T_ManWork)
rounded rectangle at (49,21)-(196,41): text "Mechanical Interlock"; invisible if NOT (NOT $Inst$.In_HomeXLock AND $Inst$.T_ManHome)
rounded rectangle at (48,42)-(122,62): text "Home"; invisible if NOT $Inst$.E_HomeErr; alarm colour if $Inst$.E_HomeErr
rounded rectangle at (122,42)-(196,62): text "Work"; invisible if NOT $Inst$.E_WorkErr; alarm colour if $Inst$.E_WorkErr
4 more shapes without text or variables
*)

(* Visualisation Std_IAI_16Point
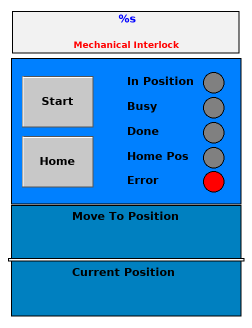
rounded rectangle at (117,58)-(193,89): text "In Position"
ellipse at (195,64)-(216,85): alarm colour if $Inst$.S_InPos
rounded rectangle at (117,83)-(193,114): text "Busy"
ellipse at (195,89)-(216,110): alarm colour if NOT $Inst$.In_PEND
rounded rectangle at (117,108)-(193,139): text "Done"
ellipse at (195,114)-(216,135): alarm colour if $Inst$.In_PEND
rounded rectangle at (117,133)-(193,164): text "Home Pos"
ellipse at (195,139)-(216,160): alarm colour if $Inst$.S_InHome
rounded rectangle at (117,157)-(193,188): text "Error"
ellipse at (195,163)-(216,184): alarm colour if .E4_Scan_IAI_Alm OR .E4_Scan_IAI_MovPos OR .E4_Scan_IAI_PosAlm
button at (14,68)-(85,119): text "Start"; taps $Inst$.T_ManStart
button at (14,128)-(85,179): text "Home"; taps $Inst$.T_ManHome
rounded rectangle at (62,193)-(175,224): text "Move To Position"
rounded rectangle at (62,249)-(175,280): text "Current Position"
rounded rectangle at (4,3)-(231,45): text "%s"; shows $Inst$.IN_Name
rounded rectangle at (45,27)-(192,47): text "Mechanical Interlock"; invisible if NOT (NOT $Inst$.In_Mec_Interlock AND ($Inst$.In_ManStart OR $Inst$.In_ManHome))
4 more shapes without text or variables
2 elements of other kinds (tables, trends, ...) not read
*)

(* Visualisation Std_IV_Vision_Ctrl
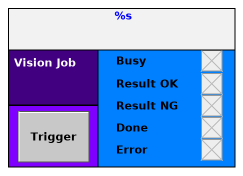
button at (10,103)-(81,154): text "Trigger"; taps $Inst$.T_ManualTrigger
rounded rectangle at (106,42)-(182,63): text "Busy"
rounded rectangle at (106,65)-(182,86): text "Result OK"
rounded rectangle at (106,109)-(182,130): text "Done"
rounded rectangle at (106,131)-(182,152): text "Error"
rounded rectangle at (106,87)-(182,108): text "Result NG"
embedded screen at (193,42)-(214,63): Green_Ind
embedded screen at (193,65)-(214,86): Green_Ind
embedded screen at (193,87)-(214,108): Red_Ind
embedded screen at (193,109)-(214,130): Green_Ind
embedded screen at (193,131)-(214,152): Red_Ind
rounded rectangle at (4,39)-(91,70): text "Vision Job"
rounded rectangle at (0,0)-(227,42): text "%s"; shows $Inst$.IN_Name
3 more shapes without text or variables
1 elements of other kinds (tables, trends, ...) not read
*)

(* Visualisation Std_Main_Ctrl_Button
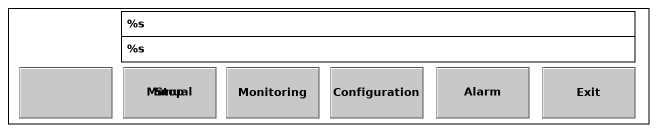
rectangle at (11,24)-(142,55): text "Message:"; invisible if NOT MC.AutoMode
rectangle at (11,-1)-(142,30): text "Machine Status:"
rectangle at (113,1)-(627,27): text "%s"; shows $Inst$.T_StatusString; alarm colour if $Inst$.T_AutoMsgAlarm
button at (218,57)-(311,108): text "Monitoring"; opens TP50_Monitoring; dynamic style cmd_ManMode
button at (322,57)-(415,108): text "Configuration"; invisible if $Inst$.InOut_SC.AutoRunning; opens TP30_PASSWORD; dynamic style cmd_ManMode
button at (428,57)-(521,108): dynamic style cmd_ManMode
rectangle at (113,26)-(627,52): text "%s"; shows T_AutoRunString; invisible if NOT MC.AutoMode
button at (534,57)-(627,108): text "Exit"; invisible if $Inst$.InOut_SC.AutoRunning; opens TP00_MAIN_EXIT; runs INTERN EXITPROGRAM; dynamic style cmd_ManMode
rectangle at (432,59)-(517,105): text "Alarm"; alarm colour if $Inst$.Out_RedTower; opens TP80_ALARM
button at (115,57)-(208,108): dynamic style cmd_ManMode
rectangle at (119,59)-(204,105): text "Manual"; invisible if MC.AutoRunning; alarm colour if MC.ManualMode; taps $Inst$.T_Manual; opens TP10_MANUAL
rectangle at (119,59)-(204,105): text "Stop"; invisible if NOT MC.AutoRunning; alarm colour if MC.StopPressed AND On_1s; taps $Inst$.T_Stop
button at (11,57)-(104,108): dynamic style btn_Auto
1 more shapes without text or variables
1 elements of other kinds (tables, trends, ...) not read
*)

(* Visualisation Std_NewPassWord
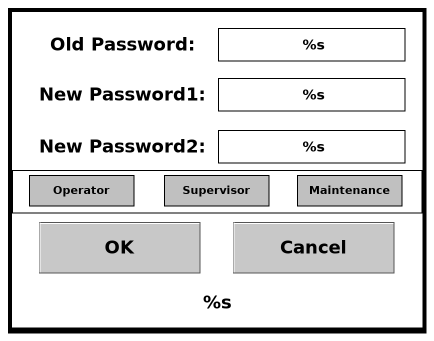
rounded rectangle at (17,20)-(206,51): text "Old Password:"; invisible if In_SelectedPasswordLvl < 2
rectangle at (207,19)-(394,52): text "%s"; shows .Password_Control.In_EntryPasswordString; invisible if In_SelectedPasswordLvl < 2; editable 0..10
button at (28,213)-(189,264): text "OK"; taps .Password_Control.In_ChangePassword
button at (222,213)-(383,264): text "Cancel"; opens TP40_SETTING
rounded rectangle at (9,278)-(404,309): text "%s"; shows .Password_Control.Out_StatusString
rounded rectangle at (17,70)-(206,101): text "New Password1:"
rectangle at (207,69)-(394,102): text "%s"; shows .Password_Control.In_NewPasswordString1; editable 0..10
rounded rectangle at (17,122)-(206,153): text "New Password2:"
rectangle at (207,121)-(394,154): text "%s"; shows .Password_Control.In_NewPasswordString2; editable 0..10
rounded rectangle at (18,166)-(123,197): text "Operator"; alarm colour if .Password_Control.In_SelectedPasswordLvl = 0; runs INTERN ASSIGN Password_Control.In_SelectedPasswordLvl:=(0)
rounded rectangle at (153,166)-(258,197): text "Supervisor"; alarm colour if .Password_Control.In_SelectedPasswordLvl = 1; runs INTERN ASSIGN Password_Control.In_SelectedPasswordLvl:=(1)
rounded rectangle at (286,166)-(391,197): text "Maintenance"; alarm colour if .Password_Control.In_SelectedPasswordLvl = 2; runs INTERN ASSIGN Password_Control.In_SelectedPasswordLvl:=(2)
3 more shapes without text or variables
3 elements of other kinds (tables, trends, ...) not read
*)

(* Visualisation Std_OnOffDev_Ctrl
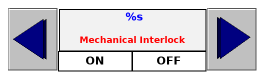
rounded rectangle at (50,0)-(197,42): text "%s"; shows $Inst$.IN_DevName
rounded rectangle at (49,42)-(123,62): text "ON"; alarm colour if $Inst$.S_OnSig
rounded rectangle at (123,42)-(197,62): text "OFF"; alarm colour if NOT $Inst$.S_OnSig
rounded rectangle at (50,21)-(197,41): text "Mechanical Interlock"; invisible if NOT (NOT $Inst$.In_OnXLock AND $Inst$.T_ManOn)
6 more shapes without text or variables
*)

(* Visualisation Std_Password
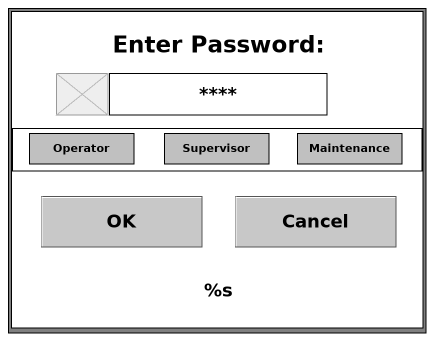
rounded rectangle at (89,20)-(330,51): text "Enter Password:"
rectangle at (100,64)-(318,106): text "****"; shows .Password_Control.In_EntryPasswordString; editable 0..10
button at (32,187)-(193,238): text "OK"; taps .Password_Control.In_EnterPassword
button at (226,187)-(387,238): text "Cancel"; opens TP00_MAIN
rounded rectangle at (89,266)-(330,297): text "%s"; shows .Password_Control.Out_StatusString
bitmap at (47,64)-(99,106): c:\flexlink\bitmap\lock.bmp
rounded rectangle at (20,124)-(125,155): text "Operator"; alarm colour if .Password_Control.In_SelectedPasswordLvl = 0; runs INTERN ASSIGN Password_Control.In_SelectedPasswordLvl:=(0)
rounded rectangle at (155,124)-(260,155): text "Supervisor"; alarm colour if .Password_Control.In_SelectedPasswordLvl = 1; runs INTERN ASSIGN Password_Control.In_SelectedPasswordLvl:=(1)
rounded rectangle at (288,124)-(393,155): text "Maintenance"; alarm colour if .Password_Control.In_SelectedPasswordLvl = 2; runs INTERN ASSIGN Password_Control.In_SelectedPasswordLvl:=(2)
3 more shapes without text or variables
3 elements of other kinds (tables, trends, ...) not read
*)

(* Visualisation Std_VacuumVal_Ctrl
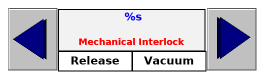
rounded rectangle at (48,0)-(195,42): text "%s"; shows $Inst$.IN_Name
rounded rectangle at (48,42)-(122,62): text "Release"; invisible if $Inst$.E_PurgeErr; alarm colour if $Inst$.S_Release
rounded rectangle at (122,42)-(196,62): text "Vacuum"; invisible if $Inst$.E_VacuumErr; alarm colour if $Inst$.S_Vacuum
group at (-2,-1)-(47,61)
  button at (0,0)-(49,62): taps $Inst$.In_ManHome
group at (197,-1)-(246,61)
  button at (0,0)-(49,61): taps $Inst$.In_ManWork
rounded rectangle at (48,23)-(195,43): text "Mechanical Interlock"; invisible if NOT (NOT $Inst$.In_VacuumX AND $Inst$.T_ManVacuum)
rounded rectangle at (48,23)-(195,43): text "Mechanical Interlock"; invisible if NOT (NOT $Inst$.In_PurgeX AND $Inst$.T_ManPurge)
rounded rectangle at (48,42)-(122,62): text "Release"; invisible if NOT $Inst$.E_PurgeErr; alarm colour if $Inst$.E_PurgeErr
rounded rectangle at (122,42)-(196,62): text "Vacuum"; invisible if NOT $Inst$.E_VacuumErr; alarm colour if $Inst$.E_VacuumErr
4 more shapes without text or variables
*)

(* Visualisation ToggleSwitch1
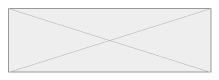
bitmap at (0,0)-(203,63): c:\flexlink\bitmap\toggleswitchgreen.bmp
bitmap at (0,0)-(203,64): c:\flexlink\bitmap\toggleswitchred.bmp
*)

(* Visualisation Yellow_Ind
